FUNCTION LimitValue : LREAL
VAR_INPUT
	Value: LREAL;
	MinValue: LREAL;
	MaxValue: LREAL;
END_VAR
VAR
  Res: LREAL;
END_VAR

Res := Value;
IF Res < MinValue THEN
	Res := MinValue;
END_IF;
IF Res > MaxValue THEN
	Res := MaxValue;
END_IF;
LimitValue := Res;

END_FUNCTION

(* stored: Version 1.1.0.1, ProductVersion 3.1.4024.3
   POU LimitValue: Id {8ec83da8-172e-4276-96b0-f8e5d7bdeff1}, SpecialFunc None *)
